(* CoDeSys 2.3 library: Standard.lib *)

(* Global variable list: Globale_Variablen *)
VAR_GLOBAL
	STANDARD_LIBVER					:	STRING(16) 	:=	'V1.20.01 Beta';	(* Version String *)
    STANDARD_MMPREADY               :   BOOL        :=  TRUE;               (* MMP Ready *)
END_VAR

(* POU CONCAT, IL *)
(******************************************************************************
Description: Concatenation of two strings
Input:
  - STR1: Source string1, after this the second is appended
  - STR2: Appended string
Output:
    none 
Return: Result string is STR1 + STR2
	If SETLARGESTRINGS(True) is called the maximum string size is 1023
    characters, otherwise the string size is limited to 255 characters.
******************************************************************************)
FUNCTION CONCAT : STRING(1023)
VAR_INPUT
	STR1:STRING(1023);
	STR2:STRING(1023);
END_VAR
LD	0
END_FUNCTION

(* POU CTD, IL *)
(******************************************************************************
Description: Counter Down
Input:
  - CD: Count Down on rising edge 
  - LOAD: Load Start Value 
  - PV: Start Value 
Output:
  - Q: Counter reached 0 
  - CV: Current Counter Value 
Return: Output is used as return value.
******************************************************************************)
FUNCTION_BLOCK CTD
VAR_INPUT
	CD: BOOL;
	LOAD: BOOL;
	PV: WORD;
END_VAR
VAR_OUTPUT
	Q: BOOL;
	CV: WORD;
END_VAR
VAR
	M: BOOL;
END_VAR
	LD		0
END_FUNCTION_BLOCK

(* POU CTU, IL *)
(******************************************************************************
Description: Counter up
Input:
  - CU: Count Up 
  - RESET: Reset Counter to 0 
  - PV: Counter Limit 
Output:
  - Q:  Counter reached the Limit 
  - CV:  Current Counter Value 
Return: Output variables are used as Return.
******************************************************************************)
FUNCTION_BLOCK CTU
VAR_INPUT
	CU: BOOL;
	RESET: BOOL;
	PV: WORD;
END_VAR
VAR_OUTPUT
	Q: BOOL;
	CV: WORD;
END_VAR
VAR
	M: BOOL;
END_VAR
LD	0
END_FUNCTION_BLOCK

(* POU CTUD, IL *)
(******************************************************************************
Description: Counter up and down
Input:
  - CU:  Count Up 
  - CD:  Count Down 
  - RESET:  Reset Counter to Null 
  - LOAD:  Load Start Value 
  - PV:  Start Value / Counter Limit 
Output:
  - QU:  Counter reached Limit 
  - QD:  Counter reached Null 
  - CV:  Current Counter Value 
Return: Output is used as return value.
******************************************************************************)
FUNCTION_BLOCK CTUD
VAR_INPUT
	CU: BOOL;
	CD: BOOL;
	RESET: BOOL;
	LOAD: BOOL;
	PV: WORD;
END_VAR
VAR_OUTPUT
	QU: BOOL;
	QD: BOOL;
	CV: WORD;
END_VAR
VAR
	MU: BOOL;
	MD: BOOL;
END_VAR
LD	0
END_FUNCTION_BLOCK

(* POU DELETE, IL *)
(******************************************************************************
Description: Deletes character of the string
Input:
  - STR: Source string
  - LEN: length of deleted sub string
  - POS: begin position of deleting
Output:
    none
Return: String without deleted substring
	If SETLARGESTRINGS(True) is called the maximum string size is 1023
    characters, otherwise the string size is limited to 255 characters.
******************************************************************************)
FUNCTION DELETE : STRING(1023)
VAR_INPUT
	STR: STRING(1023);
	LEN: INT;
	POS: INT;
END_VAR
LD	0
END_FUNCTION

(* POU LEN, IL *)
(******************************************************************************
Description: Gets length of string
Input:
  - STR: String which length is computed 
Output:
    none
Return: Length of string
******************************************************************************)
FUNCTION LEN : INT
VAR_INPUT
	STR:STRING(1023);
END_VAR
LD	0
END_FUNCTION

(* POU F_TRIG, IL *)
(******************************************************************************
Description: Falling Edge detection
Input:
  - S1:  Signal to detect 
Output:
  - Q0:  Edge detected 
Return: Output variable is used for return.
******************************************************************************)
FUNCTION_BLOCK F_TRIG
VAR_INPUT
	S1: BOOL;
END_VAR
VAR_OUTPUT
	Q0: BOOL;
END_VAR
VAR
	M: BOOL;	
END_VAR
LD	0
END_FUNCTION_BLOCK

(* POU FIND, IL *)
(******************************************************************************
Description: Find the character position of the beginning of the first 
    occurence of STR2 in STR1. 
Input:
  - STR1: String in which the substring is searched
  - STR2: Substring
Output:
    none
Return: Position in the STR1
  - 0: No occurence found
  - Else: Frst occurence of STR2 in STR1
******************************************************************************)
FUNCTION FIND : INT
VAR_INPUT
	STR1:STRING(1023);
	STR2:STRING(1023);
END_VAR
LD	0
END_FUNCTION

(* POU GETLARGESTRINGS, ST *)
(******************************************************************************
Description: Usage of large strings (up to 1023 characters) for all string
             functions
Input:
  - VAL: Pointer to return value (True or False)
Output:
  - none
Return: 0 on success, -1 on error
******************************************************************************)
FUNCTION GETLARGESTRINGS : DINT
VAR_INPUT
	VAL: POINTER TO BOOL;
END_VAR
;
END_FUNCTION

(* POU INSERT, IL *)
(******************************************************************************
Description: Insert substring at the given position
Input:
  - STR1: Sourcestring to this a substring is added
  - STR2: Substring which is added
  - POS: Position in STR1 where STR2 is added
Output:
    none
Return: Added substring
	If SETLARGESTRINGS(True) is called the maximum string size is 1023
    characters, otherwise the string size is limited to 255 characters.
******************************************************************************)
FUNCTION INSERT:STRING(1023)
VAR_INPUT
	STR1:STRING(1023);
	STR2:STRING(1023);
	POS:INT;
END_VAR
	LD		0
END_FUNCTION

(* POU LEFT, IL *)
(******************************************************************************
Description: Extracts the leftmost characters
  - STR: Soucre string
  - SIZE: count of extraction
Output:
    none
Return: Extracted string
	If SETLARGESTRINGS(True) is called the maximum string size is 1023
    characters, otherwise the string size is limited to 255 characters.
******************************************************************************)
FUNCTION LEFT : STRING(1023)
VAR_INPUT
	STR:STRING(1023);
	SIZE:INT;
END_VAR
LD	0
END_FUNCTION

(* POU MID, IL *)
(******************************************************************************
Description: Extracts substring of the source string
Input:
  - STR: Source string
  - LEN: Length of substring
  - POS: position where extraction is beginning
Output:
    none
Return: Extracted substring
	If SETLARGESTRINGS(True) is called the maximum string size is 1023
    characters, otherwise the string size is limited to 255 characters.
******************************************************************************)
FUNCTION MID : STRING(1023)
VAR_INPUT
	STR:STRING(1023);
	LEN:INT;
	POS:INT;
END_VAR
LD	0
END_FUNCTION

(* POU R_TRIG, IL *)
(******************************************************************************
Description: Rising Edge detection
Input:
  - S1:  Signal to detect 
Output:
  - Q0:  Edge detected 
Return: Output variable are used for return.
******************************************************************************)
FUNCTION_BLOCK R_TRIG
VAR_INPUT
	S1: BOOL;
END_VAR
VAR_OUTPUT
	Q0: BOOL;
END_VAR
VAR
	M: BOOL;	
END_VAR
LD	0
END_FUNCTION_BLOCK

(* POU REPLACE, IL *)
(******************************************************************************
Description: Replaces in the source string the given sub string
Input:
  - STR1: source string 
  - STR2: sub string
  - L: length of sub string
  - P: pos of source string where replacing should beginn 
Output:
    none
Return: Modified string
	If SETLARGESTRINGS(True) is called the maximum string size is 1023
    characters, otherwise the string size is limited to 255 characters.
******************************************************************************)
FUNCTION REPLACE : STRING(1023)
VAR_INPUT
	STR1:STRING(1023);
	STR2:STRING(1023);
	L:INT;
	P:INT;
END_VAR
LD	0
END_FUNCTION

(* POU RIGHT, IL *)
(******************************************************************************
Description: Extracting rightmost characters
Input:
  - STR: Source string
  - SIZE: Length of substring
Output:
    none
Return: Extracted substring
	If SETLARGESTRINGS(True) is called the maximum string size is 1023
    characters, otherwise the string size is limited to 255 characters.
******************************************************************************)
FUNCTION RIGHT : STRING(1023)
VAR_INPUT
	STR:STRING(1023);
	SIZE:INT;
END_VAR
LD	0
END_FUNCTION

(* POU RS, IL *)
(******************************************************************************
Description: Bistable function, reset dominant.
Input:
  - SET: Bistable input 
  - RESET1: Dominmant bistable input. 
Output:
  - Q1: Result of bistable function 
Return: Output variable used as return value.
******************************************************************************)
FUNCTION_BLOCK RS
VAR_INPUT
	SET: 	BOOL;
	RESET1: BOOL;
END_VAR
VAR_OUTPUT
	Q1:		BOOL;
END_VAR
LD	0
END_FUNCTION_BLOCK

(* POU RTC, IL *)
(******************************************************************************
Description: Real time clock, gets date and time. Set of date and time not 
    implemented.
Input:
  - EN:  PDT is loaded, when EN has a rising edge 
  - PDT: meaningless because set of date and time not implemented 
Output:
  - Q: A copy of EN 
  - CDT: Current date and time, valid when EN = 1 
Return: Output variables are used as return.
******************************************************************************)
FUNCTION_BLOCK RTC
VAR_INPUT
	EN:BOOL;
	PDT:DATE_AND_TIME;
END_VAR
VAR_OUTPUT
	Q:BOOL;
	CDT:DATE_AND_TIME;
END_VAR
LD 0
END_FUNCTION_BLOCK

(* POU SEMA, IL *)
(******************************************************************************
Description: Software semaphore. Interuptable!
Input:
  - CLAIM: TRUE claims Semaphore.
  - RELEASE: TRUE releases a claimed semaphore.
Output:
  - BUSY: State of Semaphore
Return: Output used as return.
  - TRUE: Semaphore is claimed
  - FALSE: Semaphore is released
******************************************************************************)
FUNCTION_BLOCK SEMA
VAR_INPUT
	CLAIM: BOOL;
	RELEASE: BOOL;
END_VAR
VAR_OUTPUT
	BUSY: BOOL;
END_VAR
VAR
	X: BOOL;
END_VAR
LD	0
END_FUNCTION_BLOCK

(* POU SETLARGESTRINGS, ST *)
(******************************************************************************
Description: Usage of large strings (up to 1023 characters) for all string
             functions
Input:
  - VAL: True or False
Output:
    none
Return: 0 on success, -1 if msys version is not compatible
******************************************************************************)
FUNCTION SETLARGESTRINGS : DINT
VAR_INPUT
	VAL: BOOL;
END_VAR
;
END_FUNCTION

(* POU SR, IL *)
(******************************************************************************
Description: Bistable function, set dominant
Input:
  - SET1: Dominant input of bistable function.
  - RESET: input of bistable function.
Output:
  - Q1: Result of Bistable function. 
Return: Output is used as return
******************************************************************************)
FUNCTION_BLOCK SR
VAR_INPUT
	SET1: BOOL;	
	RESET: BOOL;
END_VAR
VAR_OUTPUT
	Q1: BOOL;
END_VAR
LD	0
END_FUNCTION_BLOCK

(* POU Standard_GetVersion, ST *)
(******************************************************************************
Description: Returns the version string of the library. In simulation always
	'V1.00 Release' is returned.

Input:
	- dummy

Return: 
	Version String
******************************************************************************)
FUNCTION Standard_GetVersion : STRING(16)
VAR_INPUT
	dummy:	BOOL;
END_VAR
VAR
END_VAR
Standard_GetVersion := STANDARD_LIBVER;
END_FUNCTION

(* POU STCTR, IL *)
(******************************************************************************
Description: Service Time (Running Time) Counter 
 
If activated, the elapsed time between two calls is added to SERVICETIME. 
To achieve accuracy the RTC is used. If the elapsed time between two calls 
exceeds 10 sec it is not accumulated to the service time, as the RTC may have 
been adjusted. Therefore a cyclic call of at least 10 sec is required.
             
Input:
  - ACTIVE: Indicates if time counting is active 
  - RESET: Indicates if the current time counter must be set to 0
Output:
  - SERVICETIME: Currently elapsed service time (running time) in seconds. 
				 This value will be keept in RETAIN so that it can't get lost.
				 Is the sum of the time elapsed in all periods where ACTIVE
				 was set.
Return: Output is used as return value.
******************************************************************************)
FUNCTION_BLOCK STCTR
VAR_INPUT
	ACTIVE: BOOL;
	RESET: BOOL;
END_VAR
VAR_OUTPUT
	RETAIN SERVICETIME: LREAL;
END_VAR
VAR
	STARTTIME: DWORD;
END_VAR
	LD		0
END_FUNCTION_BLOCK

(* POU TOF, IL *)
(******************************************************************************
Description: Timer of delay
Input:
  - IN: Starts timer with falling edge, resets timer with rising edge 
  - PT: Time to pass, before Q is set 
Output:
  - Q: is FALSE, PT seconds after IN had a falling edge
  - ET: Elapsed time 
Return: Output variables are used for return.
******************************************************************************)
FUNCTION_BLOCK TOF
VAR_INPUT
	IN: BOOL;
	PT:TIME;
END_VAR
VAR_OUTPUT
	Q: BOOL;
	ET: TIME;
END_VAR
VAR
	M: BOOL;
	StartTime: TIME;
END_VAR
LD	0
END_FUNCTION_BLOCK

(* POU TOLOWERCASE, ST *)
(******************************************************************************
Description: convert string to lowercase. 
  - STR: Source string
Output:
    none
Return: converted string
	If SETLARGESTRINGS(True) is called the maximum string size is 1023
    characters, otherwise the string size is limited to 255 characters.
******************************************************************************)
FUNCTION TOLOWERCASE : STRING(1023)
VAR_INPUT
	STR: STRING(1023);
END_VAR
;
END_FUNCTION

(* POU TON, IL *)
(******************************************************************************
Description: Timer on delay.
Input:
  - IN: Starts timer with rising edge, resets timer with falling edge 
  - PT: Time to pass, before Q is set 
Output:
  - Q: Is TRUE, PT seconds after IN had a rising edge 
  - ET: Elapsed time 
Return: Output variables are used for return.
******************************************************************************)
FUNCTION_BLOCK TON
VAR_INPUT
	IN: BOOL;
	PT: TIME;
END_VAR
VAR_OUTPUT
	Q: BOOL;
	ET: TIME;
END_VAR
VAR
	M: BOOL;
	StartTime: TIME;	
END_VAR
LD	0
END_FUNCTION_BLOCK

(* POU TOUPPERCASE, ST *)
(******************************************************************************
Description: convert string to uppercase. 
  - STR: Source string
Output:
    none
Return: converted string
	If SETLARGESTRINGS(True) is called the maximum string size is 1023
    characters, otherwise the string size is limited to 255 characters.
******************************************************************************)
FUNCTION TOUPPERCASE : STRING(1023)
VAR_INPUT
	STR: STRING(1023);
END_VAR
;
END_FUNCTION

(* POU TP, IL *)
(******************************************************************************
Description: Timer Pulse 
Input:
  - IN: Trigger for Start of the Signal 
  - PT: The length of the High-Signal in 10ms 
Output:
  - Q: The pulse 
  - ET: The current phase of the High-Signal 
Return: Output variables are used for return.
******************************************************************************)
FUNCTION_BLOCK TP
VAR_INPUT
	IN: BOOL;
	PT: TIME;
END_VAR
VAR_OUTPUT
	Q: BOOL;
	ET: TIME;
END_VAR
VAR
	StartTime: TIME;
END_VAR
LD	0
END_FUNCTION_BLOCK

(* POU TRIM, ST *)
(******************************************************************************
Description: eliminates leading spaces and spaces at the end of the given string. 
  - STR: Source string
Output:
    none
Return: processed string
	If SETLARGESTRINGS(True) is called the maximum string size is 1023
    characters, otherwise the string size is limited to 255 characters.
******************************************************************************)
FUNCTION TRIM : STRING(1023)
VAR_INPUT
	STR: STRING(1023);
END_VAR
;
END_FUNCTION

(* POU TRIMLEFT, ST *)
(******************************************************************************
Description: eliminates leading spaces. 
  - STR: Source string
Output:
    none
Return: processed string
	If SETLARGESTRINGS(True) is called the maximum string size is 1023
    characters, otherwise the string size is limited to 255 characters.
******************************************************************************)
FUNCTION TRIMLEFT : STRING(1023)
VAR_INPUT
	STR: STRING(1023);
END_VAR
;
END_FUNCTION

(* POU TRIMRIGHT, ST *)
(******************************************************************************
Description: eliminates spaces at the end. 
  - STR: Source string
Output:
    none
Return: processed string
	If SETLARGESTRINGS(True) is called the maximum string size is 1023
    characters, otherwise the string size is limited to 255 characters.
******************************************************************************)
FUNCTION TRIMRIGHT : STRING(1023)
VAR_INPUT
	STR: STRING(1023);
END_VAR
;
END_FUNCTION
